PROGRAM Kinematics
VAR
	Fb_Axes_KinCongifGroup: FB_KinConfigGroup;
	Fb_Axes_KinResetGroup: FB_KinResetGroup;
	Fb_Axes_KinReConfigGroup: CfgReconfigGroup;
	Build_Kin_Group: TOF;
	Trig_Build: BOOL;
	bb_tp_reset: BOOL;
	BB_TP_Kin: TP;
END_VAR

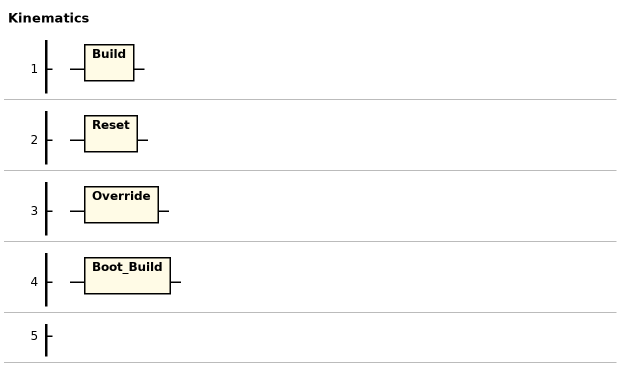
// NETWORK 1
Build();

// NETWORK 2
Reset();

// NETWORK 3
Override();

// NETWORK 4
Boot_Build();

// NETWORK 5

ACTION Boot_Build:
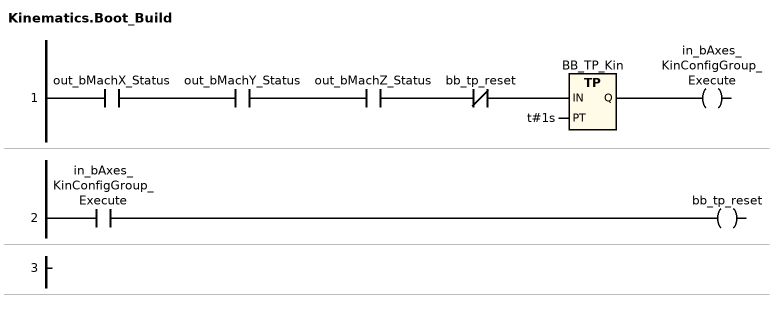
// NETWORK 1
BB_TP_Kin(IN := out_bMachX_Status AND out_bMachY_Status AND out_bMachZ_Status AND NOT bb_tp_reset, PT := t#1s); // TP
in_bAxes_KinConfigGroup_Execute := BB_TP_Kin.Q;

// NETWORK 2
bb_tp_reset := in_bAxes_KinConfigGroup_Execute;

// NETWORK 3
END_ACTION

ACTION Build:
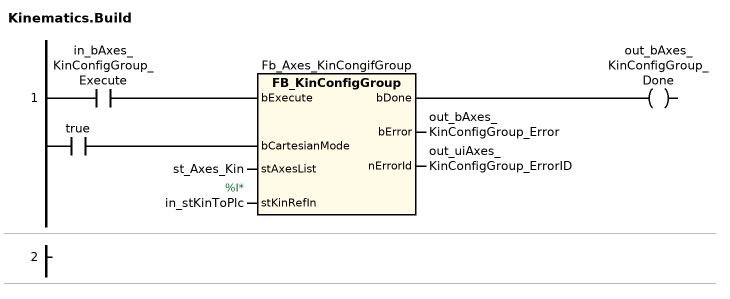
// NETWORK 1
//   in_stKinToPlc: AT %I*
Fb_Axes_KinCongifGroup(
    bExecute := in_bAxes_KinConfigGroup_Execute,
    bCartesianMode := true,
    stAxesList := st_Axes_Kin,
    stKinRefIn := in_stKinToPlc,
    bError => out_bAxes_KinConfigGroup_Error,
    nErrorId => out_uiAxes_KinConfigGroup_ErrorID); // FB_KinConfigGroup
out_bAxes_KinConfigGroup_Done := Fb_Axes_KinCongifGroup.bDone;

// NETWORK 2
END_ACTION

ACTION Override:
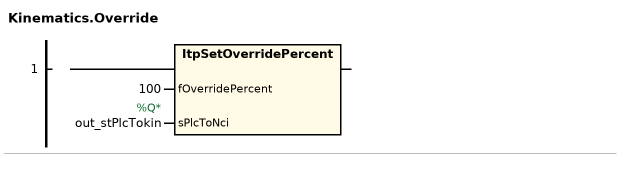
// NETWORK 1
//   out_stPlcTokin: AT %Q*
ItpSetOverridePercent(fOverridePercent := 100, sPlcToNci := out_stPlcTokin);
END_ACTION

ACTION Reset:
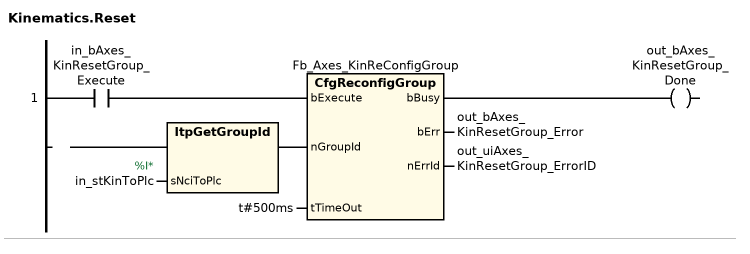
// NETWORK 1
//   in_stKinToPlc: AT %I*
Fb_Axes_KinReConfigGroup(
    bExecute := in_bAxes_KinResetGroup_Execute,
    nGroupId := ItpGetGroupId(sNciToPlc := in_stKinToPlc),
    tTimeOut := t#500ms,
    bErr => out_bAxes_KinResetGroup_Error,
    nErrId => out_uiAxes_KinResetGroup_ErrorID); // CfgReconfigGroup
out_bAxes_KinResetGroup_Done := Fb_Axes_KinReConfigGroup.bBusy;
END_ACTION

END_PROGRAM

(* stored: Version 1.1.0.1, ProductVersion 3.1.4022.17
   POU Kinematics: Id {7cb5da92-2766-494c-be1f-d28464dbc341}, SpecialFunc None
   Action Boot_Build: Id {4c718687-6cee-434d-b8a0-d865a8f08046}
   Action Build: Id {39d78f7c-fedd-41a4-989a-0c3d36f7c385}
   Action Override: Id {8d059852-d952-4778-bab3-c7e2328f4f45}
   Action Reset: Id {c91a5b4b-072c-41d4-ab20-1d1f9911e713} *)
